// TIA Portal V20 export
DATA_BLOCK "DB_Global"   // DB23
// stored: Access Published, MemoryReserve 100, Namespace Global
   VAR
      Status : Struct
         Line : Struct
            A1 : Struct
               On : Array[_.gMinA1.._.gMaxA1] of Bool;
               ReadyToRun : Array[_.gMinA1.._.gMaxA1] of Bool;
               Occupied : Array[_.gMinA1.._.gMaxA1] of Bool;
               Running : Array[_.gMinA1.._.gMaxA1] of Bool;
               Fault : Array[_.gMinA1.._.gMaxA1] of Bool;
               Estop : Array[_.gMinA1.._.gMaxA1] of Bool;
               Manual : Array[_.gMinA1.._.gMaxA1] of Bool;
               Stop : Array[_.gMinA1.._.gMaxA1] of Bool;
               Blockage : Array[_.gMinA1.._.gMaxA1] of Bool;
            END_STRUCT;
            B1 : Struct
               On : Array[_.gMinB1.._.gMaxB1] of Bool;
               ReadyToRun : Array[_.gMinB1.._.gMaxB1] of Bool;
               Occupied : Array[_.gMinB1.._.gMaxB1] of Bool;
               Running : Array[_.gMinB1.._.gMaxB1] of Bool;
               Fault : Array[_.gMinB1.._.gMaxB1] of Bool;
               Estop : Array[_.gMinB1.._.gMaxB1] of Bool;
               Manual : Array[_.gMinB1.._.gMaxB1] of Bool;
               Stop : Array[_.gMinB1.._.gMaxB1] of Bool;
               Blockage : Array[_.gMinB1.._.gMaxB1] of Bool;
            END_STRUCT;
            C1 : Struct
               On : Array[_.gMinC1.._.gMaxC1] of Bool;
               ReadyToRun : Array[_.gMinC1.._.gMaxC1] of Bool;
               Occupied : Array[_.gMinC1.._.gMaxC1] of Bool;
               Running : Array[_.gMinC1.._.gMaxC1] of Bool;
               Fault : Array[_.gMinC1.._.gMaxC1] of Bool;
               Estop : Array[_.gMinC1.._.gMaxC1] of Bool;
               Manual : Array[_.gMinC1.._.gMaxC1] of Bool;
               Stop : Array[_.gMinC1.._.gMaxC1] of Bool;
               Blockage : Array[_.gMinC1.._.gMaxC1] of Bool;
            END_STRUCT;
            D1 : Struct
               On : Array[_.gMinD1.._.gMaxD1] of Bool;
               ReadyToRun : Array[_.gMinD1.._.gMaxD1] of Bool;
               Occupied : Array[_.gMinD1.._.gMaxD1] of Bool;
               Running : Array[_.gMinD1.._.gMaxD1] of Bool;
               Fault : Array[_.gMinD1.._.gMaxD1] of Bool;
               Estop : Array[_.gMinD1.._.gMaxD1] of Bool;
               Manual : Array[_.gMinD1.._.gMaxD1] of Bool;
               Stop : Array[_.gMinD1.._.gMaxD1] of Bool;
               Blockage : Array[_.gMinD1.._.gMaxD1] of Bool;
            END_STRUCT;
         END_STRUCT;
      END_STRUCT;
   END_VAR
BEGIN
   // Status.Line.A1.On[1001] : AS1.1.1
   // Status.Line.A1.On[1002] : AS1.1.2
   // Status.Line.A1.ReadyToRun[1001] : AS1.1.1
   // Status.Line.A1.ReadyToRun[1002] : AS1.1.2
   // Status.Line.A1.Occupied[1001] : AS1.1.1
   // Status.Line.A1.Occupied[1002] : AS1.1.2
   // Status.Line.A1.Running[1001] : AS1.1.1
   // Status.Line.A1.Running[1002] : AS1.1.2
   Status.Line.A1.Fault[1001] := 0;   // AS1.1.1
   Status.Line.A1.Fault[1002] := 0;   // AS1.1.2
   Status.Line.A1.Estop[1001] := 0;   // AS1.1.1
   Status.Line.A1.Estop[1002] := 0;   // AS1.1.2
   Status.Line.A1.Manual[1001] := 0;   // AS1.1.1
   Status.Line.A1.Manual[1002] := 0;   // AS1.1.2
   Status.Line.A1.Stop[1001] := 0;   // AS1.1.1
   Status.Line.A1.Stop[1002] := 0;   // AS1.1.2
   Status.Line.A1.Blockage[1001] := 0;   // AS1.1.1
   Status.Line.A1.Blockage[1002] := 0;   // AS1.1.2
   // Status.Line.C1.ReadyToRun[3001] : BP1.1.1
   // Status.Line.C1.ReadyToRun[3002] : BP1.1.2
   // Status.Line.C1.Occupied[3001] : BP1.1.1
   // Status.Line.C1.Occupied[3002] : BP1.1.2
   // Status.Line.C1.Running[3001] : BP1.1.1
   // Status.Line.C1.Running[3002] : BP1.1.2
   // Status.Line.C1.Fault[3001] : BP1.1.1
   // Status.Line.C1.Fault[3002] : BP1.1.2
   // Status.Line.C1.Estop[3001] : BP1.1.1
   // Status.Line.C1.Estop[3002] : BP1.1.2
   // Status.Line.C1.Manual[3001] : BP1.1.1
   // Status.Line.C1.Manual[3002] : BP1.1.2
   // Status.Line.C1.Stop[3001] : BP1.1.1
   // Status.Line.C1.Stop[3002] : BP1.1.2
   // Status.Line.C1.Blockage[3001] : BP1.1.1
   // Status.Line.C1.Blockage[3002] : BP1.1.2
END_DATA_BLOCK
